KUKA KRL program: rsi_reset_pids.src, rsi_reset_pids.dat

--- rsi_reset_pids.src ---
&ACCESS RV3
DEF  RSI_RESET_PIDS ( )
   DECL INT Ret
   IF RSI_ACTIVE THEN
      Ret = rsi_setpublicpar(RSI_ID, "VIS_X_PID" , "Reset", 1)
      Ret = rsi_setpublicpar(RSI_ID, "VIS_Pos_PID" , "Reset", 1)
      Ret = rsi_setpublicpar(RSI_ID, "VIS_Height_PID" , "Reset", 1)
      Ret = rsi_setpublicpar(RSI_ID, "VIS_Dist_Height_PID" , "Reset", 1)
      Ret = rsi_setpublicpar(RSI_ID, "VIS_A_Angle_PID" , "Reset", 1)
      Ret = rsi_setpublicpar(RSI_ID, "VIS_B_Angle_PID" , "Reset", 1)
      Ret = rsi_setpublicpar(RSI_ID, "VIS_C_Angle_PID" , "Reset", 1)
   ENDIF
END

--- rsi_reset_pids.dat ---
&ACCESS RV3
DEFDAT  RSI_RESET_PIDS
;FOLD EXTERNAL DECLARATIONS;%{PE}%MKUKATPBASIS,%CEXT,%VCOMMON,%P
;FOLD BASISTECH EXT;%{PE}%MKUKATPBASIS,%CEXT,%VEXT,%P
EXT  BAS (BAS_COMMAND  :IN,REAL  :IN )
;ENDFOLD (BASISTECH EXT)
;FOLD USER EXT;%{E}%MKUKATPUSER,%CEXT,%VEXT,%P
;Make your modifications here

;ENDFOLD (USER EXT)
;ENDFOLD (EXTERNAL DECLARATIONS)
ENDDAT
